(* IEC 61131-3 sources: CodesysTest/alpha/export/ElectricMachine.dev/Plc Logic/Application/Programs, 4 files *)

(* ---- PRG_.pou.st ---- *)
(*#-#-#-#-#-#-#-#-#-#---Declaration---#-#-#-#-#-#-#-#-#-#-#-#-#*)

FUNCTION_BLOCK PRG_
VAR_INPUT
END_VAR
VAR_OUTPUT
END_VAR
VAR
END_VAR
(*#-#-#-#-#-#-#-#-#-#---Implementation---#-#-#-#-#-#-#-#-#-#-#-#-#*)

(* ---- Faults.pou.st ---- *)
(*#-#-#-#-#-#-#-#-#-#---Declaration---#-#-#-#-#-#-#-#-#-#-#-#-#*)

PROGRAM Faults
VAR
	reverseFault : FB_HMIFault;
END_VAR
(*#-#-#-#-#-#-#-#-#-#---Implementation---#-#-#-#-#-#-#-#-#-#-#-#-#*)

reverseFault(refFault := PRG_Bagger.moabHead.bagDeliverySynchronous.reverseFault);

(* ---- PRG_Bagger.pou.st ---- *)
(*#-#-#-#-#-#-#-#-#-#---Declaration---#-#-#-#-#-#-#-#-#-#-#-#-#*)

PROGRAM PRG_Bagger
VAR_INPUT

END_VAR
VAR_OUTPUT

END_VAR
VAR
	_LOTARCompleteONS : FB_ONS;
	_faulActive : BOOL;
	_faultSequenceCompleted : BOOL;
	_barcodeVerificationFailed : BOOL;
    moabHead : FB_MOABHead_Electric;
    //angledHead : FB_20degHead();
    //pneuHead : FB_PneumaticHead();
    testEIPMotor : FB_AppliedMotionStepServoEIPBase();
    faultHandler : FB_FaultHandler();
	hmiInitiate : BOOL;
	msfMotorFaults : ARRAY[0..100] OF MotorCommFault;
	numberOfMSFFaults : UINT;
	msfCommFaultONS : R_TRIG();
	msfFaultListFull : BOOL;
	festoFaults : ARRAY[0..100] OF MotorCommFault;
	numberOfFestoFaults : UINT;
	festoCommFaultONS : R_TRIG();
	festoFaultListFull : BOOL;
	currentDateAndTime : GetTime();
	resetCommFaults : BOOL;
	i : INT;
	reverseFault : FB_HMIFault := (refFault := PRG_Bagger.moabHead.bagDeliverySynchronous.reverseFault);
	faultActiveONS : FB_ONS;
	throughputCalculator : FB_Throughput();
	faultOutTimer : TON();
END_VAR
(*#-#-#-#-#-#-#-#-#-#---Implementation---#-#-#-#-#-#-#-#-#-#-#-#-#*)

//    Program: PRG_Bagger
//    Description: This program glues together the whole machine and all of its components.
//
//    Created by: Ben Hess
//    Created Date: Tuesday, April 17, 2018

moabHead();
//pneuHead();
faultHandler();
hmiInitiate := HMIData.initiateCycle;
currentDateAndTime();
//msfCommFaultONS(CLK := MSFMotor.eState <> IoDrvEthernetIP.AdapterState.RUNNING);
HMIData.bagEdgePhotoeyeCovered := NOT iBagNotPresent;
oSoftStart := TRUE;

HMIData.airFilterClean();
HMIData.pressureBarGuideShaftGuides();
HMIData.driveRollerClean();
HMIData.printHeadClean();
//HMIData.pressureBarLeak(iExtended := iPressureBarExtended, iRetracted := iPressureBarRetracted, maximumStrokeTime := (TO_REAL(HMIData.passthroughSetting / 26.6)) + 0.3);
HMIData.loadPlateLeak(iExtended := iLoadPlateExtended, iRetracted := iLoadPlateRetracted, maximumStrokeTime := 0.4);
//HMIData.msfHorizontalMotorTemp(iDriveTemp := sealFlattenerHorizontalMotorInputs[4]);
//HMIData.bagDeliveryMotorTemp(iDriveTemp := bagDeliveryMotorInputs[4]);
//HMIData.passthroughMotorTemp(iDriveTemp := jawPasstrhoughMotorInputs[4]);

IF resetCommFaults THEN
	FOR i := 0 TO numberOfMSFFaults BY 1 DO
		msfMotorFaults[i].message := '';
		msfMotorFaults[i].timeOfFault := DT#1970-1-1-1:0:0;
	END_FOR
	numberOfMSFFaults := 0;
	msfFaultListFull := FALSE;
	resetCommFaults := FALSE;
END_IF

throughputCalculator(
	inCycle:= HMIData.inCycle,
	runtimeTimeout:= ,
	reset:= HMIData.resetAverageCycleTime,
	BPM=> HMIData.calculatedCyclesPerMinute,
	BPMCycles=> ,
	BPMSeconds=> ,
	BPMIndication=> );

// HMIData.version := SVN_VERSION_INFO.VERSION;
faultOutTimer(PT := T#2S);
_LOTARCompleteONS(CLK := iPALOTAR);
IF _LOTARCompleteONS.OSF OR (moabHead.state = HEAD_STATES.Idle AND NOT iPALOTAR) THEN
	_faultSequenceCompleted := TRUE;
END_IF

// Test code to run bagger even with a barcode fault
IF ((HMIData.barcodeVerifierSelection = BCVSelection.TwoDimensional) AND (HMIData.printerSelection = LabelPrinterSelection.PrintAndApply300DPI)) THEN
	HMIData.faultActive := (_faulActive AND GlobalObjects.CollectionOfActiveFaults.faultActive AND NOT moabHead.barcodeVerificationFailed.active) OR (_faulActive AND moabHead.barcodeVerificationFailed.active AND _faultSequenceCompleted) OR (_faulActive AND GlobalObjects.CollectionOfActiveFaults.totalObj > 1);
ELSE
	HMIData.faultActive := GlobalObjects.CollectionOfActiveFaults.faultActive;
END_IF

IF GlobalObjects.CollectionOfActiveFaults.faultActive THEN
	_faulActive := TRUE;
ELSE
	_faulActive := FALSE;
	_faultSequenceCompleted := FALSE;
END_IF

//HMIData.faultActive := GlobalObjects.CollectionOfActiveFaults.faultActive;
//faultActiveONS(CLK := GlobalObjects.CollectionOfActiveFaults.faultActive);
faultActiveONS(CLK := HMIData.faultActive);
IF faultActiveONS.OSR THEN
	moabHead.hmiLight.TurnOff();
END_IF

(* ---- PRG_MainProgram.pou.st ---- *)
(*#-#-#-#-#-#-#-#-#-#---Declaration---#-#-#-#-#-#-#-#-#-#-#-#-#*)

PROGRAM PRG_MainProgram
VAR
    cycleTimeMax : TIME;
    cycleTimeMaxDINT : DINT;
    ctfb : OSCAT_BASIC.CYCLE_TIME();
	firstScanDone : BOOL;
	versionInfo : VERSION;
	saveParametersTimer : Standard.TON := (PT := T#10M);
END_VAR(*#-#-#-#-#-#-#-#-#-#---Implementation---#-#-#-#-#-#-#-#-#-#-#-#-#*)

//    Program: Main (PLC_PRG)
//    Description: This program serves as the entry point for the rest of the program
//    Created by: Ben Hess
//    Created Date: January 16th, 2018

saveParametersTimer(IN := NOT saveParametersTimer.Q AND HMIData.bagsMade.count <> 0);
IF saveParametersTimer.Q THEN
	saveParametersTimer.IN := FALSE;
	SaveValuesPeriodic();
END_IF

ctfb(ct_max => cycleTimeMax);
cycleTimeMaxDINT := TIME_TO_DINT(cycleTimeMax);
// Run other programs
PRG_Bagger();

versionInfo := GetVersion();
HMIData.version := Standard.CONCAT(TO_STRING(versionInfo.uiMajor),'.');
	BPLog.AppendToString(ADR(HMIData.version), CONCAT(TO_STRING(versionInfo.uiMinor),'.'));
	BPLog.AppendToString(ADR(HMIData.version), CONCAT(TO_STRING(versionInfo.uiServicePack),'.'));
	BPLog.AppendToString(ADR(HMIData.version), TO_STRING(versionInfo.uiPatch));
	BPLog.AppendToString(ADR(HMIData.version), TO_STRING(GetTextProperty("VersionPostfix")));

//Set maximum passthrough based on model selection
CASE HMIdata.baggerModelSelection OF
	ModelSelection.Pro18_1174,
	ModelSelection.Pro18_1183:
		 Globals.maximumPassthough := Globals.MAXIMUM_PASSTHROUGH_PRO18;

	ModelSelection.Pro24_1182,
	ModelSelection.Pro24_1196:
		 Globals.maximumPassthough := Globals.MAXIMUM_PASSTHROUGH_PRO24;
END_CASE

// Perform functions on first scan
IF NOT firstScanDone THEN
	GlobalObjects.CollectionOfLoggable.RegisterAll(internalLogger := Globals.SystemLog);
	GlobalObjects.CollectionOfInitialzable.InitializeAll();
	firstScanDone := TRUE;
	 // After first scan turn off flag set by StartDone system event
	Globals.firstScan := FALSE;
END_IF

// Start executing objects that implement IExecuteAutomatically
IF firstScanDone THEN
	GlobalObjects.CollectionOfExecutable.ExecuteAll();
	Globals.SystemLog();
END_IF

IF HMIData.ackAllFaults THEN
	GlobalObjects.CollectionOfActiveFaults.AckAll();
	HMIData.ackAllFaults := FALSE;
END_IF

//First scan flag is set by task handler and reset in main routine here
IF Globals.firstScan THEN
    Globals.firstScan := FALSE;
END_IF
